TYPE ST_RobotTaskStatusInfo :
STRUCT
	nRobotTaskStatus : WORD;
	nZoneOccupied : WORD;
	bInTask : BOOL;
	bPerformingTaskAction : BOOL;
	sRobotStatus : STRING;

END_STRUCT
END_TYPE

(* stored: Version 1.1.0.1, ProductVersion 3.1.4020.12
   DUT ST_RobotTaskStatusInfo: Id {bbf64d41-11d2-4340-b1fa-413ea3a7f148} *)
